PROGRAM MAIN
VAR
	nState: INT;
	bButon: BOOL;
	bSensor1: BOOL;
	ftrig1: F_TRIG;
	bHat: BOOL;
	rtrig1: R_TRIG;
	bSensor2: BOOL;
	random1: DRAND;
	nYukseklik: INT;
	Select1: FB_MalzemeSecme;
	T1: TON;
	T2: TON;
	T3: TON;
	bKol1: BOOL;
	bKutuSens1: BOOL;
	bKutuSens2: BOOL;
	bKutuSens3: BOOL;
	rtrig2: R_TRIG;
	rtrig3: R_TRIG;
	rtrig4: R_TRIG;
	bKol2: BOOL;
	bKol3: BOOL;
	nKisaKutu: INT;
	nOrtaKutu: INT;
	nUzunKutu: INT;
	sInfoMsg: STRING;
	sMsgKisa_1: STRING(255);
	sMsgOrta_1: STRING(255);
	sMsgUzun_1: STRING(255);
	sMsgYukseklik: STRING(255);
END_VAR


ACT_PRG();

ACT_VisuMsg();

ACTION ACT_PRG:

ftrig1(CLK:= bSensor1 , Q=> );

rtrig1(CLK:= bSensor2 , Q=> );


rtrig2(CLK:= bKutuSens1 , Q=> ); // Kısa malzeme kutusu sensörü

rtrig3(CLK:= bKutuSens2 , Q=> ); // Orta malzeme kutusu sensörü

rtrig4(CLK:= bKutuSens3 , Q=> ); // Uzun malzeme kutusu sensörü


CASE nState OF 
	

	0:
	
	IF bButon THEN 
		
		nState := 10;
		
	END_IF
	
	
	10:
	
	sInfoMsg := 'Malzeme Bekleniyor.';
	
	IF ftrig1.Q THEN
		
		nState := 20;
		
	END_IF
	
	
	20:
	
	bHat := TRUE;
	
	sInfoMsg := 'Hat Aktif, Malzemenin Konuma Gelmesi Bekleniyor.';

	IF rtrig1.Q THEN
		
		bHat := FALSE;
		
		random1(Seed:=10 , Num=> );
		nYukseklik := LREAL_TO_INT(random1.Num * 100);
		
		nState := 30;
		
	END_IF
	
	
	30:
		
	Select1(nValue:=nYukseklik,
			nStateOut=>nState, 
			sMsg =>sInfoMsg );	
	
	
	32:
	
		bHat := TRUE;
		T1(IN:=TRUE , PT:=T#2S);
		
		IF T1.Q THEN
			nState := 42;
			T1(IN:=FALSE);
			bHat := FALSE;
		END_IF
	
	34:
	
		bHat := TRUE;
		T2(IN:=TRUE , PT:=T#4S);
		
		IF T2.Q THEN
			nState := 44;
			T2(IN:=FALSE);
			bHat := FALSE;
		END_IF
	
	
	36:
		bHat := TRUE;
		T3(IN:=TRUE , PT:=T#6S);
		
		IF T3.Q THEN
			nState := 46;
			T3(IN:=FALSE);
			bHat := FALSE;
		END_IF
		
		
	42:
		
		bKol1 := TRUE;
		sInfoMsg	:=	'Kısa Boyutlu Malzeme Kutusuna Koyuluyor.';
		
		IF rtrig2.Q THEN
			
			bKol1 := FALSE;
			
			nKisaKutu := nKisakutu + 1;
			
			nState := 0;
			
		END_IF
		
		
	
	44:
	
		bKol2 := TRUE;
		sInfoMsg	:=	'Orta Boyutlu Malzeme Kutusuna Koyuluyor.';
		
		IF rtrig3.Q THEN
			
			bKol2 := FALSE;
			
			nOrtaKutu := nOrtaKutu + 1;
			
			nState := 0;
			
		END_IF	

	46:
		bKol3:= TRUE;
		sInfoMsg	:=	'Uzun Boyutlu Malzeme Kutusuna Koyuluyor.';
		
		IF rtrig4.Q THEN
			
			bKol3 := FALSE;
			
			nUzunKutu := nUzunKutu + 1;
			
			nState := 0;
			
		END_IF	
	
			
END_CASE


	IF NOT bButon THEN 
		
		nState := 0;
		sInfoMsg := 'Sistem Kapali.';
		bKol1 := FALSE;
		bKol2 := FALSE;
		bKol3 := FALSE;
		T1(IN:=FALSE);
		T2(IN:=FALSE);
		T3(IN:=FALSE);
		
	END_IF
END_ACTION

ACTION ACT_VisuMsg:


sMsgKisa_1 := CONCAT(STR1:='Kisa Malzeme Kutusunda ' , STR2:= INT_TO_STRING(nKisaKutu) );
sMsgKisa_1 := CONCAT(STR1:=sMsgKisa_1 , STR2:= ' Malzeme Var' );

sMsgOrta_1 := CONCAT(STR1:='Orta Malzeme Kutusunda ' , STR2:= INT_TO_STRING(nOrtaKutu) );
sMsgOrta_1 := CONCAT(STR1:=sMsgOrta_1 , STR2:= ' Malzeme Var' );

sMsgUzun_1 := CONCAT(STR1:='Uzun Malzeme Kutusunda ' , STR2:= INT_TO_STRING(nUzunKutu) );
sMsgUzun_1 := CONCAT(STR1:=sMsgUzun_1 , STR2:= ' Malzeme Var' );

sMsgYukseklik := CONCAT(STR1:='Malzeme Yüksekligi: ' , STR2:= INT_TO_STRING(nYukseklik) );
sMsgYukseklik := CONCAT(STR1:=sMsgYukseklik , STR2:= ' [cm]' );
END_ACTION

END_PROGRAM

(* stored: Version 1.1.0.1, ProductVersion 3.1.4024.4
   POU MAIN: Id {80ee3623-f28a-44be-b20d-920e9e8fec7c}, SpecialFunc None
   Action ACT_PRG: Id {343a227b-6950-40dc-a3d2-f8760d16042a}
   Action ACT_VisuMsg: Id {0c989fe7-d8ef-4545-bff2-357eb7051986} *)
